(*********************************** G.D S.p.A. - Technical Department ***********************************
============= PROGRAM INFO ============
FOLDER:             TBD
MACHINES INVOLVED:  TBD 

============= DESCRIPTION =============
csp main interface program

============= REVISIONS ===============
Date		Version	 	Author      	Description             
----------	-------		------------  	--------------------------------------------
2019/09/27 	0000.00	 	M.Grasso		Creation of the PRG

**********************************************************************************************************)
PROGRAM _csp_case_discharge_normal
VAR
END_VAR

(* CASE *)
	(* DISCHARGE *)
		(* SPEEDBELT *)
		csp_case_discharge_speedBelt();
		(* REJECT *)
		csp_case_discharge_reject();

END_PROGRAM

(* stored: Version 1.1.0.1, ProductVersion 3.1.4024.3
   POU _csp_case_discharge_normal: Id {26e4d132-b279-47db-9c6e-d269cfa6b3b5}, SpecialFunc None *)
